// Mitsubishi GX Works2 project: connection_2   PLC: Q03UDV

PROGRAM MAIN
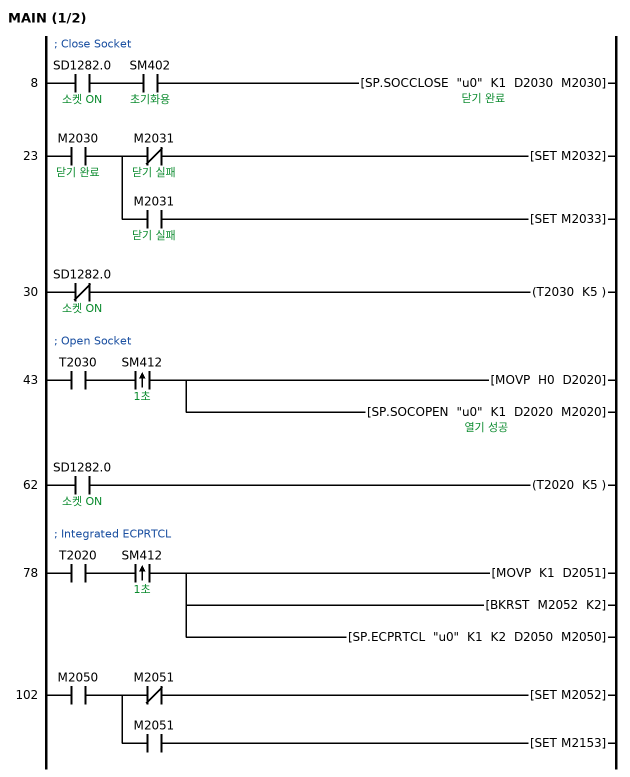
; Close Socket
8     LD      SD1282.0  ; 소켓 ON
      AND     SM402  ; 초기화용
      SP.SOCCLOSE "u0" K1 D2030 M2030  ; 닫기 완료
23    LD      M2030  ; 닫기 완료
      MPS
      ANI     M2031  ; 닫기 실패
      SET     M2032
      MPP
      AND     M2031  ; 닫기 실패
      SET     M2033
30    LDI     SD1282.0  ; 소켓 ON
      OUT     T2030 K5
; Open Socket
43    LD      T2030
      ANDP    SM412  ; 1초
      MOVP    H0 D2020
      SP.SOCOPEN "u0" K1 D2020 M2020  ; 열기 성공
62    LD      SD1282.0  ; 소켓 ON
      OUT     T2020 K5
; Integrated ECPRTCL
78    LD      T2020
      ANDP    SM412  ; 1초
      MOVP    K1 D2051
      BKRST   M2052 K2
      SP.ECPRTCL "u0" K1 K2 D2050 M2050
102   LD      M2050
      MPS
      ANI     M2051
      SET     M2052
      MPP
      AND     M2051
      SET     M2153
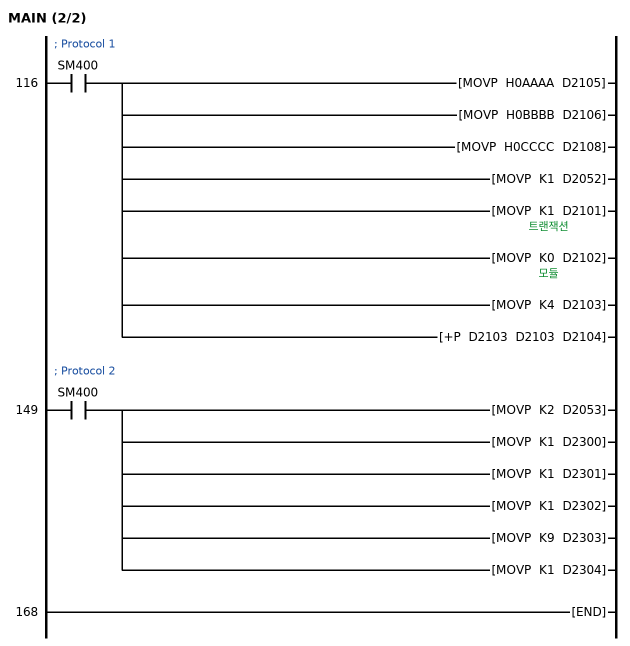
; Protocol 1
116   LD      SM400
      MOVP    H0AAAA D2105
      MOVP    H0BBBB D2106
      MOVP    H0CCCC D2108
      MOVP    K1 D2052
      MOVP    K1 D2101  ; 트랜잭션
      MOVP    K0 D2102  ; 모듈
      MOVP    K4 D2103
      +P      D2103 D2103 D2104
; Protocol 2
149   LD      SM400
      MOVP    K2 D2053
      MOVP    K1 D2300
      MOVP    K1 D2301
      MOVP    K1 D2302
      MOVP    K9 D2303
      MOVP    K1 D2304
168   END
END_PROGRAM

// device comments not shown above
M2100  ; 통신 성공
M2101  ; 통신 실패
M2300  ; 읽기 성공
M2301  ; 읽기 실패
D2152  ; 리퀘스트
